{attribute 'Tc2GvlVarNames'}
VAR_GLOBAL CONSTANT
	(* Regelventil_Zustand_Status *)
	E_RV_Zustand_Status_Idle_Sperre			: SINT := 0;
	E_RV_Zustand_Status_Betriebsbereit		: SINT := 1;
	E_RV_Zustand_Status_Nachl				: SINT := 2;
	E_RV_Zustand_Status_Vorl				: SINT := 3;
	E_RV_Zustand_Status_Betrieb				: SINT := 4;
	E_RV_Zustand_Status_Betrieb_Sperre		: SINT := 5;
	E_RV_Zustand_Status_Stoerung			: SINT := 99;

	(* Regelventil_Zustand_Regelung_Modus *)
	E_RV_Regelung_Modus_Stellung			: SINT := 0;
	E_RV_Regelung_Modus_Temp_Heizen			: SINT := 1;
	E_RV_Regelung_Modus_Temp_Kuehlen		: SINT := 2;
END_VAR

(* stored: Version 1.1.0.1, ProductVersion 3.1.4024.9
   GVL Con_RV: Id {d627ebfe-37fa-44e3-a82f-a576125d723a} *)
